{attribute 'qualified_only'}
{attribute 'strict'}
TYPE eTcoToggleTaskTests :
(
    Reinit := 1001,
    CleanUp := 1002,
    Message := 1003,
    TriggerToggleWhileRunNotCalled := 1004,
    TriggerToggleWhileDisabled := 1005,
    TriggerToggleWhileEnabled := 1006,
    TriggerOnWhileRunNotCalled := 1007,
    TriggerOnWhileDisabled := 1008,
    TriggerOnWhileEnabled := 1009,
    TriggerOffWhileRunNotCalled := 1010,
    TriggerOffWhileDisabled := 1011,
    TriggerOffWhileEnabled := 1012
);
END_TYPE

(* stored: Version 1.1.0.1
   DUT eTcoToggleTaskTests: Id {9d986438-740b-0107-34c5-afef7aa116f2} *)
